// TIA Portal project "Move" (V16)

(* hardware
DEVICE "S7-1200 station_1"  S7-1200 Station
   slot 0: "Rack_0"  S7-1200 Rack  Rack  V1.0
   slot 1: "PLC_1"  CPU 1214C AC/DC/Rly  6ES7 214-1BG40-0XB0  V4.4
*)

// ===== PLC "PLC_1"  CPU 1214C AC/DC/Rly =====

VAR_GLOBAL   // PLC tag table "Tabla de variables estándar"
   "Tag_1" AT %I0.1 : Bool;
   "Tag_2" AT %I0.2 : Bool;
   "Tag_3" AT %I0.3 : Bool;
   "Tag_4" AT %I0.4 : Bool;
   "Tag_5" AT %MW105 : Int;
   "Tag_6" AT %MD106 : DWord;
   "Tag_7" AT %MD115 : DWord;
   "Tag_8" AT %MD120 : Time;
   "Tag_9" AT %I0.5 : Bool;
   "Tag_10" AT %I0.6 : Bool;
   "Tag_11" AT %MD130 : Time;
   "Tag_12" AT %Q0.1 : Bool;
END_VAR

// folder: System blocks/Program resources

DATA_BLOCK "IEC_Counter_0_DB_1"   // DB2
{ S7_Optimized_Access := 'TRUE' }
AUTHOR : Simatic
FAMILY : IEC
NAME : CNTR
VERSION : 1.0
// stored: InstanceOfName IEC_COUNTER
"IEC_COUNTER"
BEGIN
END_DATA_BLOCK

DATA_BLOCK "IEC_Timer_0_DB_1"   // DB4
{ S7_Optimized_Access := 'TRUE' }
AUTHOR : Simatic
FAMILY : IEC
NAME : IEC_TMR
VERSION : 1.0
// stored: InstanceOfName IEC_TIMER
"IEC_TIMER"
BEGIN
END_DATA_BLOCK

// folder: (top level)

ORGANIZATION_BLOCK "Main"   // OB1, LAD, ProgramCycle
TITLE = "Main Program Sweep (Cycle)"
{ S7_Optimized_Access := 'TRUE' }
VERSION : 0.1
   VAR_INPUT
      Initial_Call : Bool;   // Initial call of this OB
      Remanence : Bool;   // =True, if remanent data are available
   END_VAR
BEGIN

REGION Network 1
   // El Move transfiere el contenido de entrada a una dirección de memoria.
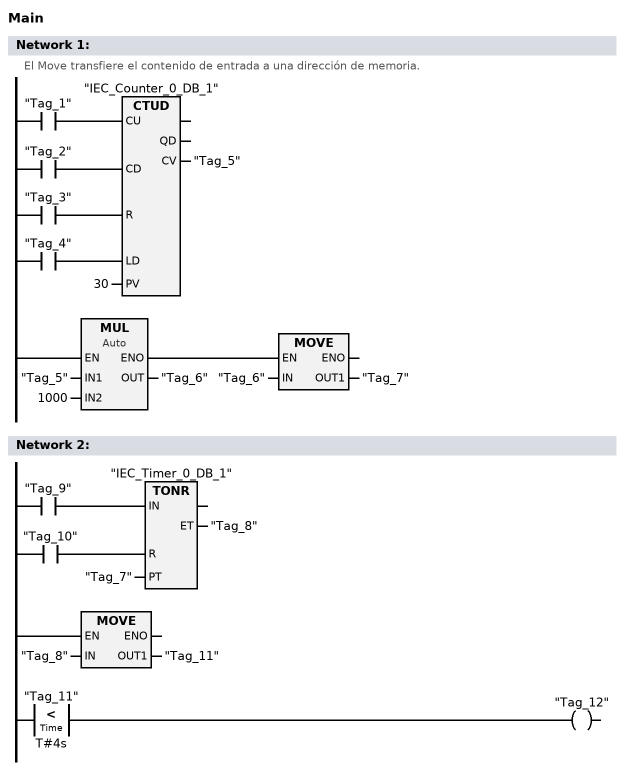
   "IEC_Counter_0_DB_1".CTUD(CU := "Tag_1", CD := "Tag_2", R := "Tag_3", LD := "Tag_4", PV := 30, CV => "Tag_5");
   "Tag_6" := "Tag_5" * 1000;
   "Tag_7" := "Tag_6";
END_REGION

REGION Network 2
   "IEC_Timer_0_DB_1".TONR(IN := "Tag_9", R := "Tag_10", PT := "Tag_7", ET => "Tag_8");
   "Tag_11" := "Tag_8";
   "Tag_12" := "Tag_11" < T#4s;
END_REGION
END_ORGANIZATION_BLOCK